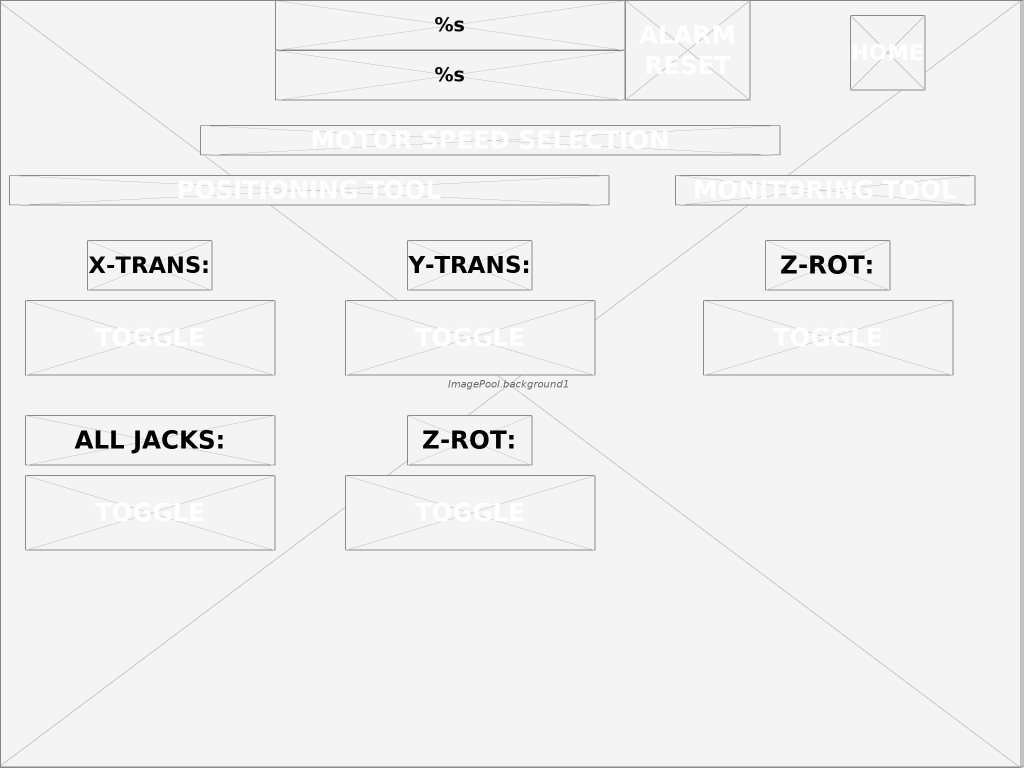
VISUALIZATION MOTOR_SPEEDS_SCREEN  // 1024x768
    Image (-3,0 1024x768), image: ImagePool.background1
    Image (200,125 580x30), "MOTOR SPEED SELECTION", image: VisuDialogs.ImagePoolDialogs.Title2
    Image (625,0 125x100), "ALARM RESET", image: ImagePool.PB_BU_125_100
        p84334746: MAIN.Visualization.P00B_Alarm_Reset.bitmap_ID
        OnMouseDown: execute { MAIN.Visualization.P00B_Alarm_Reset.Active:=TRUE; }
        OnMouseUp: execute { MAIN.Visualization.P00B_Alarm_Reset.Active:=FALSE; }
    Image (275,0 350x50), "%s", text variable: MAIN.Visualization.P00D_Station_Status.display_text, image: ImagePool.IN_BU_300_50
        p84334746: MAIN.Visualization.P00D_Station_Status.bitmap_ID
    Image (275,50 350x50), "%s", text variable: MAIN.Visualization.P00D_Alarm_Status.display_text, image: ImagePool.IN_BU_300_50
        p84334746: MAIN.Visualization.P00D_Alarm_Status.bitmap_ID
    Image (9,175 600x30), "POSITIONING TOOL", image: VisuDialogs.ImagePoolDialogs.Title2
    Image (675,175 300x30), "MONITORING TOOL", image: VisuDialogs.ImagePoolDialogs.Title
    Image (25,415 250x50), "ALL JACKS:", image: ImagePool.IN_CL_300_50
    Image (25,300 250x75), "TOGGLE", image: ImagePool.PB_BU_250_75
        OnMouseDown: execute { MAIN.Visualization.P13B_TRANSX_SPEED_Toggle.Active := TRUE; }
        OnMouseUp: execute { MAIN.Visualization.P13B_TRANSX_SPEED_Toggle.Active := FALSE; }
    Image (87,240 125x50), "X-TRANS:", image: ImagePool.IN_CL_300_50
    Image (345,300 250x75), "TOGGLE", image: ImagePool.PB_BU_250_75
        OnMouseDown: execute { MAIN.Visualization.P13B_TRANSY_SPEED_Toggle.Active := TRUE; }
        OnMouseUp: execute { MAIN.Visualization.P13B_TRANSY_SPEED_Toggle.Active := FALSE; }
    Image (407,240 125x50), "Y-TRANS:", image: ImagePool.IN_CL_300_50
    Image (25,475 250x75), "TOGGLE", image: ImagePool.PB_BU_250_75
        OnMouseDown: execute { MAIN.Visualization.P13B_All_JACKS_SPEED_Toggle.Active := TRUE; }
        OnMouseUp: execute { MAIN.Visualization.P13B_All_JACKS_SPEED_Toggle.Active := FALSE; }
    Image (345,475 250x75), "TOGGLE", image: ImagePool.PB_BU_250_75
        OnMouseDown: execute { MAIN.Visualization.P13B_POS_TOOL_ZROT_SPEED_Toggle.Active := TRUE; }
        OnMouseUp: execute { MAIN.Visualization.P13B_POS_TOOL_ZROT_SPEED_Toggle.Active := FALSE; }
    Image (407,415 125x50), "Z-ROT:", image: ImagePool.IN_CL_300_50
    Image (765,240 125x50), "Z-ROT:", image: ImagePool.IN_CL_300_50
    Image (703,300 250x75), "TOGGLE", image: ImagePool.PB_BU_250_75
        OnMouseDown: execute { MAIN.Visualization.P13B_MON_TOOL_ZROT_SPEED_Toggle.Active := TRUE; }
        OnMouseUp: execute { MAIN.Visualization.P13B_MON_TOOL_ZROT_SPEED_Toggle.Active := FALSE; }
    Image (850,15 75x75), "HOME", image: ImagePool.PB_BU_75_75
        OnMouseDown: execute { MAIN.Visualization.P13B_HOME_SCREEN.Active := TRUE; }
        OnMouseUp: execute { MAIN.Visualization.P13B_HOME_SCREEN.Active := FALSE; }
END_VISUALIZATION

(* stored: Version 1.1.0.1, ProductVersion 3.1.4024.0
   Visu MOTOR_SPEEDS_SCREEN: Id {b3a7bd25-6697-45df-9d0f-638cec2d7052} *)
